// TIA Portal V19 export
DATA_BLOCK "A01_Config"   // DB17
// stored: MemoryReserve 100
   VAR RETAIN
      Area01_Main { ExternalAccessible := 'False'; ExternalVisible := 'False'; ExternalWritable := 'False'} : "AreaConfig";
      CoilHandlingMatCounter { ExternalAccessible := 'False'; ExternalVisible := 'False'; ExternalWritable := 'False'} : Struct
         Default_FAK { S7_SetPoint := 'True'} : LReal := 1.00109822;
      END_STRUCT;
      CoilHandling { ExternalAccessible := 'False'; ExternalVisible := 'False'; ExternalWritable := 'False'} : "CoilHandling_Config";
      Coilcar { ExternalAccessible := 'False'; ExternalVisible := 'False'; ExternalWritable := 'False'} : Struct
         LsStopDelayON : Time := T#100MS;
         LsStopDelayOFF : Time := T#100MS;
         Move : "SpeedMachine_Config";
         Lift1 : "ValveMachine_Config";
         Lift2 : "ValveMachine_Config";
      END_STRUCT;
      Area01_HU { ExternalAccessible := 'False'; ExternalVisible := 'False'; ExternalWritable := 'False'} : Struct
         Pump { S7_SetPoint := 'True'} : "HU_Pump_Config";
         Tank { S7_SetPoint := 'True'} : "HU_Tank_Config";
      END_STRUCT;
      Decoiler_HU { ExternalAccessible := 'False'; ExternalVisible := 'False'; ExternalWritable := 'False'} : Struct
         Pump { S7_SetPoint := 'True'} : "HU_Pump_Config";
         Tank { S7_SetPoint := 'True'} : "HU_Tank_Config";
      END_STRUCT;
      DecoilersHRot { ExternalAccessible := 'False'; ExternalVisible := 'False'; ExternalWritable := 'False'} : Struct
         Rotation : "ValveMachine_Config";
         Pivot : "ValveMachine_Config";
         Traslation : "Positioning_DOL_Machine_Config";
      END_STRUCT;
      Decoiler_1_2 { ExternalAccessible := 'False'; ExternalVisible := 'False'; ExternalWritable := 'False'} : Struct
         Loop : Struct
            Exist_S_MinHigh : Bool := FALSE;
            Exist_S_SpeedAdjust : Bool := TRUE;
         END_STRUCT;
         Feed : "SpeedMachine_Config";
         Jaws : "ValveMachine_Config";
         Coupling : "ValveMachine_Config";
         SnubberLift : "ValveMachine_Config";
         SnubberRoll : "ValveMachine_Config";
         Enable_End_Of_Coil_Using_Loop : Bool := FALSE;
      END_STRUCT;
      Peeler { ExternalAccessible := 'False'; ExternalVisible := 'False'; ExternalWritable := 'False'} : Struct
         Lift : "ValveMachine_Config";
         Extension : "ValveMachine_Config";
      END_STRUCT;
      Straightener { ExternalAccessible := 'False'; ExternalVisible := 'False'; ExternalWritable := 'False'} : Struct
         Feed : "PositioningMachine_Config";
         Lift_Entry : "ValveMachine_Config";
         Lift_Exit : "ValveMachine_Config";
         Lift_Entry_Exist : Bool := TRUE;
         Lift_Exit_Exist : Bool := FALSE;
      END_STRUCT;
      JB { ExternalAccessible := 'False'; ExternalVisible := 'False'; ExternalWritable := 'False'} : Struct
         MeasurePasslineReference : Real := 404.5;   // Distance of sheet passline from reference
         MaxMaterialWidth : Real := 400.0;
         Torch : "Positioning_DOL_Machine_Config";
         ClampEntry : "ValveMachine_Config";
         ClampExit : "ValveMachine_Config";
         CutHead : "ValveMachine_Config";
         Pinchroll_Feed : "SpeedMachine_Config";
         Pinchroll_Lift : "ValveMachine_Config";
      END_STRUCT;
      Loop1 { ExternalAccessible := 'False'; ExternalVisible := 'False'; ExternalWritable := 'False'} : Struct
         PitTables_Exist : Bool := TRUE;
         Entry_PercentagePosError : LReal := 95.0;   // % Max Delta Counter position Vs Positions calculated from velocity
         Exit_PercentagePosError : LReal := 95.0;   // % Max Delta Counter position Vs Positions calculated from velocity
         Delay_CheckNoEntryBkwEnable : Time := T#6S;
         Delay_CheckNoEntryFwdEnable : Time := T#6S;
         Delay_CheckNoExitBkwEnable : Time := T#6S;
         Delay_CheckNoExitFwdEnable : Time := T#6S;
      END_STRUCT;
   END_VAR
BEGIN
   Area01_Main.TimeOutStopImmediate := T#2S;
   Area01_Main.TimeOutStopInPhase := T#5S;
   Area01_Main.TimeOutStopProgrammed := T#5M;
   Area01_Main.TimeOutResetAlarms := T#1S;
   CoilHandling.SensorsDelayOn := T#250MS;
   CoilHandling.SensorsDelayOff := T#250MS;
   CoilHandling.CoilDiameterSetLoopSynchro := 510.0;
   CoilHandling.CoilDiameterRstLoopSynchro := 600.0;
   CoilHandling.MatCounter_Exist := TRUE;
   Coilcar.Move.SLS_VEL := 5000.0;
   Coilcar.Move.DelayMissingCondition := T#3S;
   Coilcar.Move.Ax.SINA_Drive.ReferenceVelocity := 2200.0;
   Coilcar.Move.Ax.SINA_Drive.InvertDirection := FALSE;
   Coilcar.Move.Ax.MinAccTime := 0.1;
   Coilcar.Move.Ax.MinDecTime := 0.1;
   Coilcar.Move.Ax.LeadScrewPitchVal := 490.088453;
   Coilcar.Move.Ax.MotorRevolution := 198.0;
   Coilcar.Move.Ax.LoadRevolution := 1.0;
   Coilcar.Move.Ax.PowerOffDelay := T#5S;
   Coilcar.Move.Ax.StandstillVelocity := 50.0;
   Coilcar.Move.Ax.StandstillDelay := T#200MS;
   Coilcar.Move.Fan.Presence := FALSE;
   Coilcar.Move.Fan.DelayOff := T#0MS;
   Coilcar.Move.Brake_Presence := FALSE;
   Coilcar.Lift1.DelayPressureRunningTimeout := T#3S;
   Coilcar.Lift1.DelayMissingCondition := T#3S;
   Coilcar.Lift1.Rest_LsQty := 1;
   Coilcar.Lift1.Work_LsQty := 1;
   Coilcar.Lift1.Rest_RetainAut := FALSE;
   Coilcar.Lift1.Work_RetainAut := FALSE;
   Coilcar.Lift1.V.RestLimSwitchExist := FALSE;
   Coilcar.Lift1.V.WorkLimSwitchExist := TRUE;
   Coilcar.Lift1.V.CheckOilInPressure := TRUE;
   Coilcar.Lift1.V.CutRestWhenIsAtRest := FALSE;
   Coilcar.Lift1.V.CutWorkWhenIsAtWork := FALSE;
   Coilcar.Lift1.V.RestTime := T#5S;
   Coilcar.Lift1.V.WorkTime := T#1MS;
   Coilcar.Lift1.V.RestTimeOut := T#1H;
   Coilcar.Lift1.V.WorkTimeOut := T#1H;
   Coilcar.Lift2.DelayPressureRunningTimeout := T#3S;
   Coilcar.Lift2.DelayMissingCondition := T#3S;
   Coilcar.Lift2.Rest_LsQty := 1;
   Coilcar.Lift2.Work_LsQty := 1;
   Coilcar.Lift2.Rest_RetainAut := FALSE;
   Coilcar.Lift2.Work_RetainAut := FALSE;
   Coilcar.Lift2.V.RestLimSwitchExist := TRUE;
   Coilcar.Lift2.V.WorkLimSwitchExist := FALSE;
   Coilcar.Lift2.V.CheckOilInPressure := TRUE;
   Coilcar.Lift2.V.CutRestWhenIsAtRest := FALSE;
   Coilcar.Lift2.V.CutWorkWhenIsAtWork := FALSE;
   Coilcar.Lift2.V.RestTime := T#1MS;
   Coilcar.Lift2.V.WorkTime := T#5S;
   Coilcar.Lift2.V.RestTimeOut := T#1H;
   Coilcar.Lift2.V.WorkTimeOut := T#1H;
   Area01_HU.Pump.SafetyCutOffValveExist := TRUE;
   Area01_HU.Pump.StandbyValveExist := TRUE;
   Area01_HU.Pump.OilPumpContactotFeedbackTimeOut := T#250MS;
   Area01_HU.Tank.RecirculationPumpExist := FALSE;
   Area01_HU.Tank.HeatExchangerFanExist := FALSE;
   Area01_HU.Tank.HeatingUnitExistNum := 0;
   Area01_HU.Tank.ChillerExist := FALSE;
   Area01_HU.Tank.OilMaxTemperature := 70.0;
   Area01_HU.Tank.WaterMaxTemperature := 60.0;
   Area01_HU.Tank.TemperatureStartCheckFilters := 35.0;
   Area01_HU.Tank.HeatingHysteresys := 1.0;
   Area01_HU.Tank.DelayHeatingStart := T#30S;
   Area01_HU.Tank.DelayHeatingStop := T#30S;
   Area01_HU.Tank.DelayCollingStart := T#30S;
   Area01_HU.Tank.DelayCollingStop := T#30S;
   Area01_HU.Tank.AnlOilTemp_HighLimit := 100.0;
   Area01_HU.Tank.AnlOilTemp_LowLimit := 0.0;
   Area01_HU.Tank.AnlWaterTemp_HighLimit := 100.0;
   Area01_HU.Tank.AnlWaterTemp_LowLimit := -10.0;
   Decoiler_HU.Pump.SafetyCutOffValveExist := FALSE;
   Decoiler_HU.Pump.StandbyValveExist := TRUE;
   Decoiler_HU.Pump.OilPumpContactotFeedbackTimeOut := T#250MS;
   Decoiler_HU.Tank.RecirculationPumpExist := FALSE;
   Decoiler_HU.Tank.HeatExchangerFanExist := FALSE;
   Decoiler_HU.Tank.HeatingUnitExistNum := 0;
   Decoiler_HU.Tank.ChillerExist := FALSE;
   Decoiler_HU.Tank.OilMaxTemperature := 70.0;
   Decoiler_HU.Tank.WaterMaxTemperature := 60.0;
   Decoiler_HU.Tank.TemperatureStartCheckFilters := 35.0;
   Decoiler_HU.Tank.HeatingHysteresys := 1.0;
   Decoiler_HU.Tank.DelayHeatingStart := T#30S;
   Decoiler_HU.Tank.DelayHeatingStop := T#30S;
   Decoiler_HU.Tank.DelayCollingStart := T#30S;
   Decoiler_HU.Tank.DelayCollingStop := T#30S;
   Decoiler_HU.Tank.AnlOilTemp_HighLimit := 100.0;
   Decoiler_HU.Tank.AnlOilTemp_LowLimit := 0.0;
   Decoiler_HU.Tank.AnlWaterTemp_HighLimit := 100.0;
   Decoiler_HU.Tank.AnlWaterTemp_LowLimit := -10.0;
   DecoilersHRot.Rotation.DelayPressureRunningTimeout := T#3S;
   DecoilersHRot.Rotation.DelayMissingCondition := T#3S;
   DecoilersHRot.Rotation.Rest_LsQty := 1;
   DecoilersHRot.Rotation.Work_LsQty := 1;
   DecoilersHRot.Rotation.Rest_RetainAut := FALSE;
   DecoilersHRot.Rotation.Work_RetainAut := FALSE;
   DecoilersHRot.Rotation.V.RestLimSwitchExist := TRUE;
   DecoilersHRot.Rotation.V.WorkLimSwitchExist := TRUE;
   DecoilersHRot.Rotation.V.CheckOilInPressure := TRUE;
   DecoilersHRot.Rotation.V.CutRestWhenIsAtRest := TRUE;
   DecoilersHRot.Rotation.V.CutWorkWhenIsAtWork := TRUE;
   DecoilersHRot.Rotation.V.RestTime := T#500MS;
   DecoilersHRot.Rotation.V.WorkTime := T#500MS;
   DecoilersHRot.Rotation.V.RestTimeOut := T#1H;
   DecoilersHRot.Rotation.V.WorkTimeOut := T#1H;
   DecoilersHRot.Pivot.DelayPressureRunningTimeout := T#3S;
   DecoilersHRot.Pivot.DelayMissingCondition := T#3S;
   DecoilersHRot.Pivot.Rest_LsQty := 1;
   DecoilersHRot.Pivot.Work_LsQty := 1;
   DecoilersHRot.Pivot.Rest_RetainAut := FALSE;
   DecoilersHRot.Pivot.Work_RetainAut := FALSE;
   DecoilersHRot.Pivot.V.RestLimSwitchExist := TRUE;
   DecoilersHRot.Pivot.V.WorkLimSwitchExist := TRUE;
   DecoilersHRot.Pivot.V.CheckOilInPressure := TRUE;
   DecoilersHRot.Pivot.V.CutRestWhenIsAtRest := TRUE;
   DecoilersHRot.Pivot.V.CutWorkWhenIsAtWork := TRUE;
   DecoilersHRot.Pivot.V.RestTime := T#1MS;
   DecoilersHRot.Pivot.V.WorkTime := T#1MS;
   DecoilersHRot.Pivot.V.RestTimeOut := T#1H;
   DecoilersHRot.Pivot.V.WorkTimeOut := T#1H;
   DecoilersHRot.Traslation.DelayMissingCondition := T#3S;
   DecoilersHRot.Traslation.CyclicOBTime_ms := 0.0;
   DecoilersHRot.Traslation.Ax.limitMinus := 0.0;
   DecoilersHRot.Traslation.Ax.limitPlus := 0.0;
   DecoilersHRot.Traslation.Ax.Backlash := 0.0;
   DecoilersHRot.Traslation.Ax.BacklashActivation := FALSE;
   DecoilersHRot.Traslation.Ax.ToleranceWindow := 0.1;
   DecoilersHRot.Traslation.Ax.ToleranceWindowDelay := T#100MS;
   DecoilersHRot.Traslation.Ax.PreCutOff := 0.0;
   DecoilersHRot.Traslation.Ax.PreEndLowSpeed := 0.0;
   DecoilersHRot.Traslation.Ax.PreEndMedSpeed := 0.0;
   DecoilersHRot.Traslation.Ax.ChangeDirectionDelay := T#0MS;
   DecoilersHRot.Traslation.Ax.StandstillVelocity := 0.5;
   DecoilersHRot.Traslation.Ax.StandStillDelay := T#100MS;
   DecoilersHRot.Traslation.Ax.HomingDirection := FALSE;
   DecoilersHRot.Traslation.Ax.RecallTime := 0.0;
   DecoilersHRot.Traslation.Ax.VelocityFilter_T := 10.0;
   DecoilersHRot.Traslation.Ax.VelocityMeasUnit := 2;
   DecoilersHRot.Traslation.Ax.PosFbkDisabled := FALSE;
   DecoilersHRot.Traslation.Ax.FbkCtrlDisabled := TRUE;
   DecoilersHRot.Traslation.Ax_UM2."m" := 1.0;
   DecoilersHRot.Traslation.Ax_UM2.q := 0.0;
   DecoilersHRot.Traslation.S120.SpeedMotor.ReferenceVelocity := 2200.0;
   DecoilersHRot.Traslation.S120.SpeedMotor.InvertDirection := FALSE;
   DecoilersHRot.Traslation.S120.PowerOffDelay := T#5S;
   DecoilersHRot.Traslation.S120.StandstillVelocity := 50.0;
   DecoilersHRot.Traslation.S120.AccTime := 0.25;
   DecoilersHRot.Traslation.S120.DecTime := 0.25;
   DecoilersHRot.Traslation.Fan.Presence := FALSE;
   DecoilersHRot.Traslation.Fan.DelayOff := T#10M;
   DecoilersHRot.Traslation.Brake_Presence := FALSE;
   Decoiler_1_2.Feed.SLS_VEL := 5000.0;
   Decoiler_1_2.Feed.DelayMissingCondition := T#3S;
   Decoiler_1_2.Feed.Ax.SINA_Drive.ReferenceVelocity := 2200.0;
   Decoiler_1_2.Feed.Ax.SINA_Drive.InvertDirection := FALSE;
   Decoiler_1_2.Feed.Ax.MinAccTime := 0.1;
   Decoiler_1_2.Feed.Ax.MinDecTime := 0.1;
   Decoiler_1_2.Feed.Ax.LeadScrewPitchVal := 0.0;
   Decoiler_1_2.Feed.Ax.MotorRevolution := 10125.0;
   Decoiler_1_2.Feed.Ax.LoadRevolution := 100.0;
   Decoiler_1_2.Feed.Ax.PowerOffDelay := T#5S;
   Decoiler_1_2.Feed.Ax.StandstillVelocity := 50.0;
   Decoiler_1_2.Feed.Ax.StandstillDelay := T#200MS;
   Decoiler_1_2.Feed.Fan.Presence := TRUE;
   Decoiler_1_2.Feed.Fan.DelayOff := T#1M;
   Decoiler_1_2.Feed.Brake_Presence := FALSE;
   Decoiler_1_2.Jaws.DelayPressureRunningTimeout := T#3S;
   Decoiler_1_2.Jaws.DelayMissingCondition := T#3S;
   Decoiler_1_2.Jaws.Rest_LsQty := 1;
   Decoiler_1_2.Jaws.Work_LsQty := 1;
   Decoiler_1_2.Jaws.Rest_RetainAut := FALSE;
   Decoiler_1_2.Jaws.Work_RetainAut := FALSE;
   Decoiler_1_2.Jaws.V.RestLimSwitchExist := FALSE;
   Decoiler_1_2.Jaws.V.WorkLimSwitchExist := FALSE;
   Decoiler_1_2.Jaws.V.CheckOilInPressure := TRUE;
   Decoiler_1_2.Jaws.V.CutRestWhenIsAtRest := FALSE;
   Decoiler_1_2.Jaws.V.CutWorkWhenIsAtWork := FALSE;
   Decoiler_1_2.Jaws.V.RestTime := T#500MS;
   Decoiler_1_2.Jaws.V.WorkTime := T#500MS;
   Decoiler_1_2.Jaws.V.RestTimeOut := T#1H;
   Decoiler_1_2.Jaws.V.WorkTimeOut := T#1H;
   Decoiler_1_2.Coupling.DelayPressureRunningTimeout := T#3S;
   Decoiler_1_2.Coupling.DelayMissingCondition := T#3S;
   Decoiler_1_2.Coupling.Rest_LsQty := 1;
   Decoiler_1_2.Coupling.Work_LsQty := 1;
   Decoiler_1_2.Coupling.Rest_RetainAut := FALSE;
   Decoiler_1_2.Coupling.Work_RetainAut := FALSE;
   Decoiler_1_2.Coupling.V.RestLimSwitchExist := TRUE;
   Decoiler_1_2.Coupling.V.WorkLimSwitchExist := TRUE;
   Decoiler_1_2.Coupling.V.CheckOilInPressure := TRUE;
   Decoiler_1_2.Coupling.V.CutRestWhenIsAtRest := FALSE;
   Decoiler_1_2.Coupling.V.CutWorkWhenIsAtWork := FALSE;
   Decoiler_1_2.Coupling.V.RestTime := T#500MS;
   Decoiler_1_2.Coupling.V.WorkTime := T#500MS;
   Decoiler_1_2.Coupling.V.RestTimeOut := T#1H;
   Decoiler_1_2.Coupling.V.WorkTimeOut := T#1H;
   Decoiler_1_2.SnubberLift.DelayPressureRunningTimeout := T#3S;
   Decoiler_1_2.SnubberLift.DelayMissingCondition := T#3S;
   Decoiler_1_2.SnubberLift.Rest_LsQty := 1;
   Decoiler_1_2.SnubberLift.Work_LsQty := 1;
   Decoiler_1_2.SnubberLift.Rest_RetainAut := FALSE;
   Decoiler_1_2.SnubberLift.Work_RetainAut := FALSE;
   Decoiler_1_2.SnubberLift.V.RestLimSwitchExist := TRUE;
   Decoiler_1_2.SnubberLift.V.WorkLimSwitchExist := FALSE;
   Decoiler_1_2.SnubberLift.V.CheckOilInPressure := TRUE;
   Decoiler_1_2.SnubberLift.V.CutRestWhenIsAtRest := FALSE;
   Decoiler_1_2.SnubberLift.V.CutWorkWhenIsAtWork := FALSE;
   Decoiler_1_2.SnubberLift.V.RestTime := T#1S;
   Decoiler_1_2.SnubberLift.V.WorkTime := T#1S;
   Decoiler_1_2.SnubberLift.V.RestTimeOut := T#1H;
   Decoiler_1_2.SnubberLift.V.WorkTimeOut := T#1H;
   Decoiler_1_2.SnubberRoll.DelayPressureRunningTimeout := T#3S;
   Decoiler_1_2.SnubberRoll.DelayMissingCondition := T#3S;
   Decoiler_1_2.SnubberRoll.Rest_LsQty := 1;
   Decoiler_1_2.SnubberRoll.Work_LsQty := 1;
   Decoiler_1_2.SnubberRoll.Rest_RetainAut := FALSE;
   Decoiler_1_2.SnubberRoll.Work_RetainAut := FALSE;
   Decoiler_1_2.SnubberRoll.V.RestLimSwitchExist := FALSE;
   Decoiler_1_2.SnubberRoll.V.WorkLimSwitchExist := FALSE;
   Decoiler_1_2.SnubberRoll.V.CheckOilInPressure := TRUE;
   Decoiler_1_2.SnubberRoll.V.CutRestWhenIsAtRest := FALSE;
   Decoiler_1_2.SnubberRoll.V.CutWorkWhenIsAtWork := FALSE;
   Decoiler_1_2.SnubberRoll.V.RestTime := T#1S;
   Decoiler_1_2.SnubberRoll.V.WorkTime := T#1S;
   Decoiler_1_2.SnubberRoll.V.RestTimeOut := T#1H;
   Decoiler_1_2.SnubberRoll.V.WorkTimeOut := T#1H;
   Peeler.Lift.DelayPressureRunningTimeout := T#3S;
   Peeler.Lift.DelayMissingCondition := T#3S;
   Peeler.Lift.Rest_LsQty := 1;
   Peeler.Lift.Work_LsQty := 1;
   Peeler.Lift.Rest_RetainAut := FALSE;
   Peeler.Lift.Work_RetainAut := FALSE;
   Peeler.Lift.V.RestLimSwitchExist := TRUE;
   Peeler.Lift.V.WorkLimSwitchExist := TRUE;
   Peeler.Lift.V.CheckOilInPressure := TRUE;
   Peeler.Lift.V.CutRestWhenIsAtRest := TRUE;
   Peeler.Lift.V.CutWorkWhenIsAtWork := TRUE;
   Peeler.Lift.V.RestTime := T#500MS;
   Peeler.Lift.V.WorkTime := T#1S;
   Peeler.Lift.V.RestTimeOut := T#1H;
   Peeler.Lift.V.WorkTimeOut := T#1H;
   Peeler.Extension.DelayPressureRunningTimeout := T#3S;
   Peeler.Extension.DelayMissingCondition := T#3S;
   Peeler.Extension.Rest_LsQty := 1;
   Peeler.Extension.Work_LsQty := 1;
   Peeler.Extension.Rest_RetainAut := FALSE;
   Peeler.Extension.Work_RetainAut := FALSE;
   Peeler.Extension.V.RestLimSwitchExist := TRUE;
   Peeler.Extension.V.WorkLimSwitchExist := FALSE;
   Peeler.Extension.V.CheckOilInPressure := TRUE;
   Peeler.Extension.V.CutRestWhenIsAtRest := TRUE;
   Peeler.Extension.V.CutWorkWhenIsAtWork := FALSE;
   Peeler.Extension.V.RestTime := T#500MS;
   Peeler.Extension.V.WorkTime := T#500MS;
   Peeler.Extension.V.RestTimeOut := T#1H;
   Peeler.Extension.V.WorkTimeOut := T#1H;
   Straightener.Feed.SLS_VEL := 6000.0;
   Straightener.Feed.DelayMissingCondition := T#3S;
   Straightener.Feed.Ax.OptionON_EncoderSelection := FALSE;
   Straightener.Feed.Ax.OptionON_ParameterChange := FALSE;
   Straightener.Feed.Ax.OptionON_AutoReloadPosition := TRUE;
   Straightener.Feed.Ax.OptionON_ManPreset := FALSE;
   Straightener.Feed.Ax.HomeMode := 0;
   Straightener.Feed.Ax.PosAxis.Simulation := FALSE;
   Straightener.Feed.Ax.PosAxis.PowerOffDelay := T#10S;
   Straightener.Feed.Ax.PosAxis.PowerStartMode := 1;
   Straightener.Feed.Ax.PosAxis.PowerStopMode := 2;
   Straightener.Feed.Fan.Presence := TRUE;
   Straightener.Feed.Fan.DelayOff := T#1M;
   Straightener.Feed.Brake_Presence := FALSE;
   Straightener.Lift_Entry.DelayPressureRunningTimeout := T#10S;
   Straightener.Lift_Entry.DelayMissingCondition := T#3S;
   Straightener.Lift_Entry.Rest_LsQty := 1;
   Straightener.Lift_Entry.Work_LsQty := 1;
   Straightener.Lift_Entry.Rest_RetainAut := FALSE;
   Straightener.Lift_Entry.Work_RetainAut := FALSE;
   Straightener.Lift_Entry.V.RestLimSwitchExist := TRUE;
   Straightener.Lift_Entry.V.WorkLimSwitchExist := FALSE;
   Straightener.Lift_Entry.V.CheckOilInPressure := FALSE;
   Straightener.Lift_Entry.V.CutRestWhenIsAtRest := FALSE;
   Straightener.Lift_Entry.V.CutWorkWhenIsAtWork := FALSE;
   Straightener.Lift_Entry.V.RestTime := T#1MS;
   Straightener.Lift_Entry.V.WorkTime := T#250MS;
   Straightener.Lift_Entry.V.RestTimeOut := T#1H;
   Straightener.Lift_Entry.V.WorkTimeOut := T#1H;
   Straightener.Lift_Exit.DelayPressureRunningTimeout := T#10S;
   Straightener.Lift_Exit.DelayMissingCondition := T#3S;
   Straightener.Lift_Exit.Rest_LsQty := 1;
   Straightener.Lift_Exit.Work_LsQty := 1;
   Straightener.Lift_Exit.Rest_RetainAut := FALSE;
   Straightener.Lift_Exit.Work_RetainAut := FALSE;
   Straightener.Lift_Exit.V.RestLimSwitchExist := FALSE;
   Straightener.Lift_Exit.V.WorkLimSwitchExist := FALSE;
   Straightener.Lift_Exit.V.CheckOilInPressure := FALSE;
   Straightener.Lift_Exit.V.CutRestWhenIsAtRest := FALSE;
   Straightener.Lift_Exit.V.CutWorkWhenIsAtWork := FALSE;
   Straightener.Lift_Exit.V.RestTime := T#2S;
   Straightener.Lift_Exit.V.WorkTime := T#2S;
   Straightener.Lift_Exit.V.RestTimeOut := T#1H;
   Straightener.Lift_Exit.V.WorkTimeOut := T#1H;
   JB.Torch.DelayMissingCondition := T#3S;
   JB.Torch.CyclicOBTime_ms := 10.0;
   JB.Torch.Ax.limitMinus := 0.0;
   JB.Torch.Ax.limitPlus := 0.0;
   JB.Torch.Ax.Backlash := 0.0;
   JB.Torch.Ax.BacklashActivation := FALSE;
   JB.Torch.Ax.ToleranceWindow := 0.1;
   JB.Torch.Ax.ToleranceWindowDelay := T#100MS;
   JB.Torch.Ax.PreCutOff := 0.0;
   JB.Torch.Ax.PreEndLowSpeed := 0.0;
   JB.Torch.Ax.PreEndMedSpeed := 0.0;
   JB.Torch.Ax.ChangeDirectionDelay := T#0MS;
   JB.Torch.Ax.StandstillVelocity := 0.5;
   JB.Torch.Ax.StandStillDelay := T#100MS;
   JB.Torch.Ax.HomingDirection := FALSE;
   JB.Torch.Ax.RecallTime := 0.0;
   JB.Torch.Ax.VelocityFilter_T := 10.0;
   JB.Torch.Ax.VelocityMeasUnit := 2;
   JB.Torch.Ax.PosFbkDisabled := FALSE;
   JB.Torch.Ax.FbkCtrlDisabled := TRUE;
   JB.Torch.Ax_UM2."m" := 1.0;
   JB.Torch.Ax_UM2.q := 0.0;
   JB.Torch.S120.SpeedMotor.ReferenceVelocity := 2200.0;
   JB.Torch.S120.SpeedMotor.InvertDirection := FALSE;
   JB.Torch.S120.PowerOffDelay := T#5S;
   JB.Torch.S120.StandstillVelocity := 50.0;
   JB.Torch.S120.AccTime := 0.25;
   JB.Torch.S120.DecTime := 0.25;
   JB.Torch.Fan.Presence := FALSE;
   JB.Torch.Fan.DelayOff := T#10M;
   JB.Torch.Brake_Presence := FALSE;
   JB.ClampEntry.DelayPressureRunningTimeout := T#3S;
   JB.ClampEntry.DelayMissingCondition := T#3S;
   JB.ClampEntry.Rest_LsQty := 1;
   JB.ClampEntry.Work_LsQty := 1;
   JB.ClampEntry.Rest_RetainAut := FALSE;
   JB.ClampEntry.Work_RetainAut := FALSE;
   JB.ClampEntry.V.RestLimSwitchExist := TRUE;
   JB.ClampEntry.V.WorkLimSwitchExist := FALSE;
   JB.ClampEntry.V.CheckOilInPressure := FALSE;
   JB.ClampEntry.V.CutRestWhenIsAtRest := FALSE;
   JB.ClampEntry.V.CutWorkWhenIsAtWork := FALSE;
   JB.ClampEntry.V.RestTime := T#1MS;
   JB.ClampEntry.V.WorkTime := T#250MS;
   JB.ClampEntry.V.RestTimeOut := T#1H;
   JB.ClampEntry.V.WorkTimeOut := T#1H;
   JB.ClampExit.DelayPressureRunningTimeout := T#3S;
   JB.ClampExit.DelayMissingCondition := T#3S;
   JB.ClampExit.Rest_LsQty := 1;
   JB.ClampExit.Work_LsQty := 1;
   JB.ClampExit.Rest_RetainAut := FALSE;
   JB.ClampExit.Work_RetainAut := FALSE;
   JB.ClampExit.V.RestLimSwitchExist := TRUE;
   JB.ClampExit.V.WorkLimSwitchExist := FALSE;
   JB.ClampExit.V.CheckOilInPressure := FALSE;
   JB.ClampExit.V.CutRestWhenIsAtRest := FALSE;
   JB.ClampExit.V.CutWorkWhenIsAtWork := FALSE;
   JB.ClampExit.V.RestTime := T#1MS;
   JB.ClampExit.V.WorkTime := T#250MS;
   JB.ClampExit.V.RestTimeOut := T#1H;
   JB.ClampExit.V.WorkTimeOut := T#1H;
   JB.CutHead.DelayPressureRunningTimeout := T#3S;
   JB.CutHead.DelayMissingCondition := T#3S;
   JB.CutHead.Rest_LsQty := 1;
   JB.CutHead.Work_LsQty := 1;
   JB.CutHead.Rest_RetainAut := FALSE;
   JB.CutHead.Work_RetainAut := FALSE;
   JB.CutHead.V.RestLimSwitchExist := TRUE;
   JB.CutHead.V.WorkLimSwitchExist := TRUE;
   JB.CutHead.V.CheckOilInPressure := TRUE;
   JB.CutHead.V.CutRestWhenIsAtRest := FALSE;
   JB.CutHead.V.CutWorkWhenIsAtWork := FALSE;
   JB.CutHead.V.RestTime := T#1MS;
   JB.CutHead.V.WorkTime := T#1MS;
   JB.CutHead.V.RestTimeOut := T#1H;
   JB.CutHead.V.WorkTimeOut := T#1H;
   JB.Pinchroll_Feed.SLS_VEL := 5000.0;
   JB.Pinchroll_Feed.DelayMissingCondition := T#3S;
   JB.Pinchroll_Feed.Ax.SINA_Drive.ReferenceVelocity := 2200.0;
   JB.Pinchroll_Feed.Ax.SINA_Drive.InvertDirection := FALSE;
   JB.Pinchroll_Feed.Ax.MinAccTime := 0.1;
   JB.Pinchroll_Feed.Ax.MinDecTime := 0.1;
   JB.Pinchroll_Feed.Ax.LeadScrewPitchVal := 314.159265;
   JB.Pinchroll_Feed.Ax.MotorRevolution := 795.0;
   JB.Pinchroll_Feed.Ax.LoadRevolution := 10.0;
   JB.Pinchroll_Feed.Ax.PowerOffDelay := T#0MS;
   JB.Pinchroll_Feed.Ax.StandstillVelocity := 50.0;
   JB.Pinchroll_Feed.Ax.StandstillDelay := T#100MS;
   JB.Pinchroll_Feed.Fan.Presence := FALSE;
   JB.Pinchroll_Feed.Fan.DelayOff := T#0MS;
   JB.Pinchroll_Feed.Brake_Presence := FALSE;
   JB.Pinchroll_Lift.DelayPressureRunningTimeout := T#3S;
   JB.Pinchroll_Lift.DelayMissingCondition := T#3S;
   JB.Pinchroll_Lift.Rest_LsQty := 1;
   JB.Pinchroll_Lift.Work_LsQty := 1;
   JB.Pinchroll_Lift.Rest_RetainAut := FALSE;
   JB.Pinchroll_Lift.Work_RetainAut := FALSE;
   JB.Pinchroll_Lift.V.RestLimSwitchExist := TRUE;
   JB.Pinchroll_Lift.V.WorkLimSwitchExist := FALSE;
   JB.Pinchroll_Lift.V.CheckOilInPressure := FALSE;
   JB.Pinchroll_Lift.V.CutRestWhenIsAtRest := FALSE;
   JB.Pinchroll_Lift.V.CutWorkWhenIsAtWork := FALSE;
   JB.Pinchroll_Lift.V.RestTime := T#1MS;
   JB.Pinchroll_Lift.V.WorkTime := T#250MS;
   JB.Pinchroll_Lift.V.RestTimeOut := T#1H;
   JB.Pinchroll_Lift.V.WorkTimeOut := T#1H;
END_DATA_BLOCK
